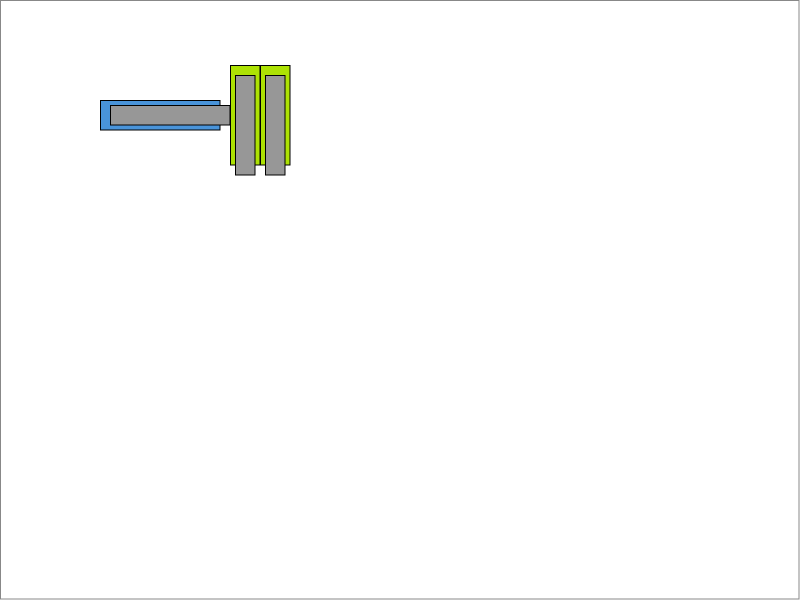
VISUALIZATION VISU_ST110  // 800x600
    Rectangle (100,100 120x30)
    Rectangle (110,105 120x20)
        p3560616238: GVL._Process2.fb_Pnp.fb_simu_axis110_01Y.rOUT_PixActual
    Rectangle (230,65 30x100)
        p3560616238: GVL._Process2.fb_Pnp.fb_simu_axis110_01Y.rOUT_PixActual
    Rectangle (235,75 20x100)
        p2738717112: GVL._Process2.fb_Pnp.fb_simu_axis110_02Z.rOUT_PixActual
        p3560616238: GVL._Process2.fb_Pnp.fb_simu_axis110_01Y.rOUT_PixActual
    Rectangle (260,65 30x100)
        p3560616238: GVL._Process2.fb_Pnp.fb_simu_axis110_01Y.rOUT_PixActual
    Rectangle (265,75 20x100)
        p2738717112: GVL._Process2.fb_Pnp.fb_simu_axis110_03Z.rOUT_PixActual
        p3560616238: GVL._Process2.fb_Pnp.fb_simu_axis110_01Y.rOUT_PixActual
END_VISUALIZATION

(* stored: Version 1.1.0.1, ProductVersion 3.1.4024.6
   Visu VISU_ST110: Id {e87517ac-fb2f-4d50-b21f-e5c3a310ec53} *)
